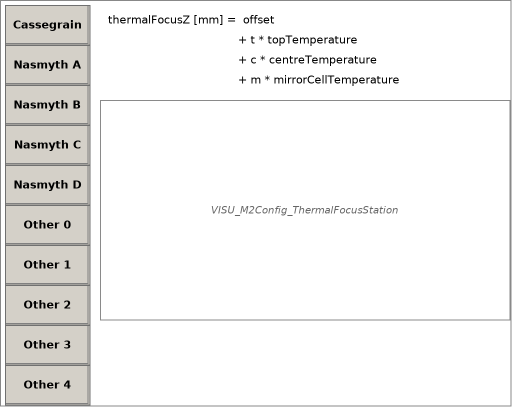
VISUALIZATION VISU_M2Config_ThermalFocus  // 512x407
VAR_IN_OUT
	currentPosition : INT;
    editable : M2ThermalFocusConfig;
	active : M2ThermalFocusConfig;
END_VAR
    Label (105,5 350x30), "thermalFocusZ [mm] = offset"
    Button (5,5 85x40), "Cassegrain", pressed state: currentPosition = 0
        OnMouseClick: execute { currentPosition := 0; }
    Button (5,45 85x40), "Nasmyth A", pressed state: currentPosition = 1
        OnMouseClick: execute { currentPosition := 1; }
    Button (5,85 85x40), "Nasmyth B", pressed state: currentPosition = 2
        OnMouseClick: execute { currentPosition := 2; }
    Button (5,125 85x40), "Nasmyth C", pressed state: currentPosition = 3
        OnMouseClick: execute { currentPosition := 3; }
    Button (5,165 85x40), "Nasmyth D", pressed state: currentPosition = 4
        OnMouseClick: execute { currentPosition := 4; }
    Button (5,205 85x40), "Other 0", pressed state: currentPosition = 5
        OnMouseClick: execute { currentPosition := 5; }
    Button (5,245 85x40), "Other 1", pressed state: currentPosition = 6
        OnMouseClick: execute { currentPosition := 6; }
    Button (5,285 85x40), "Other 2", pressed state: currentPosition = 7
        OnMouseClick: execute { currentPosition := 7; }
    Button (5,325 85x40), "Other 3", pressed state: currentPosition = 8
        OnMouseClick: execute { currentPosition := 8; }
    Button (5,365 85x40), "Other 4", pressed state: currentPosition = 9
        OnMouseClick: execute { currentPosition := 9; }
    Label (235,25 225x30), "+ t * topTemperature"
    Label (235,45 205x30), "+ c * centreTemperature"
    Label (235,65 220x30), "+ m * mirrorCellTemperature"
    Frame (100,100 410x220), frame switch variable: currentPosition
        shows VISU_M2Config_ThermalFocusStation(editable := editable.cassegrain, active := active.cassegrain)
        shows VISU_M2Config_ThermalFocusStation(editable := editable.nasmythA, active := active.nasmythA)
        shows VISU_M2Config_ThermalFocusStation(editable := editable.nasmythB, active := active.nasmythB)
        shows VISU_M2Config_ThermalFocusStation(editable := editable.nasmythC, active := active.nasmythC)
        shows VISU_M2Config_ThermalFocusStation(editable := editable.nasmythD, active := active.nasmythD)
        shows VISU_M2Config_ThermalFocusStation(editable := editable.other0, active := active.other0)
        shows VISU_M2Config_ThermalFocusStation(editable := editable.other1, active := active.other1)
        shows VISU_M2Config_ThermalFocusStation(editable := editable.other2, active := active.other2)
        shows VISU_M2Config_ThermalFocusStation(editable := editable.other3, active := active.other3)
        shows VISU_M2Config_ThermalFocusStation(editable := editable.other4, active := active.other4)
        shows VISU_M3Config_KnownPosition(active := active.position9)
END_VISUALIZATION

(* stored: Version 1.1.0.1, ProductVersion 3.1.4019.2
   Visu VISU_M2Config_ThermalFocus: Id {7905cb62-f10f-4e1a-9af9-361fbc2535f9} *)
